SUBAPPLICATION rastend (* Subapplication Type *)
  (* Standard: 61499-2; Description: Copyright (c) 2024 Meisterschulen am Ostbahnhof This program and the accompanying materials are made available under the terms of the Eclipse Public License 2.0 which is available at https://www.eclipse.org/legal/epl-2.0/ SPDX-License-Identifier: EPL-2.0 *)
  (* Version 1.0, 2024-10-23, Franz Höpfinger, Meisterschulen am Ostbahnhof *)
  PACKAGE MyLib::sys;
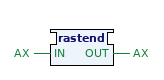
  SOCKETS
    IN : adapter::types::unidirectional::AX;
  END_SOCKETS
  PLUGS
    OUT : adapter::types::unidirectional::AX;
  END_PLUGS
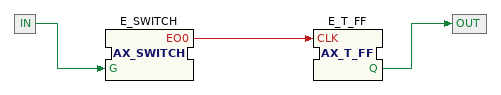
  (* soll beim Loslassen gestarte t werden ! *)
  FBS
    E_T_FF : adapter::events::unidirectional::AX_T_FF;
    E_SWITCH : adapter::events::unidirectional::AX_SWITCH;
  END_FBS
  EVENT_CONNECTIONS
    E_SWITCH.EO0 TO E_T_FF.CLK;
  END_CONNECTIONS
  ADAPTER_CONNECTIONS
    IN TO E_SWITCH.G;
    E_T_FF.Q TO OUT;
  END_CONNECTIONS
END_SUBAPPLICATION
